Omron CX-Programmer project NewProject (CX-Programmer 9.73)

# PLC NewPLC1: CP1E N20

## Global symbols (name address type ; comment)
0.01 BOOL  ; pb start
0.02 BOOL  ; relay
100.01 BOOL  ; LAMP 1
100.02 BOOL  ; LAMP 2
100.03 BOOL  ; LAMP 3
100.04 BOOL  ; LAMP4
C001 BOOL  ; COUNTER
T001 BOOL  ; TIMER
T002 BOOL  ; TIMER 2
T003 BOOL  ; TIMER 3

## Program NewProgram1 (cyclic task 0)

### Section Section1

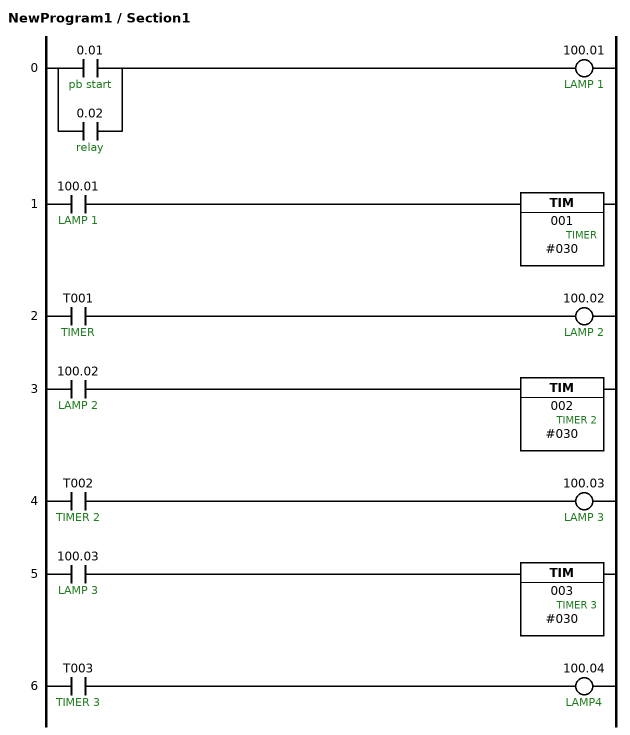
; rung 0
LD 0.01  ; pb start
OR 0.02  ; relay
OUT 100.01  ; LAMP 1
; rung 1
LD 100.01  ; LAMP 1
TIM 001 #030  ; TIMER
; rung 2
LD T001  ; TIMER
OUT 100.02  ; LAMP 2
; rung 3
LD 100.02  ; LAMP 2
TIM 002 #030  ; TIMER 2
; rung 4
LD T002  ; TIMER 2
OUT 100.03  ; LAMP 3
; rung 5
LD 100.03  ; LAMP 3
TIM 003 #030  ; TIMER 3
; rung 6
LD T003  ; TIMER 3
OUT 100.04  ; LAMP4

### Section END
; rung 0
END(001)